METHOD FINAL metSave : BOOL
VAR_INPUT
    itfDataTypeObj  :   ITF_DATATYPE;
END_VAR
VAR
    uiSafetyCount   :   UINT;
    wPos            :   WORD;
    xSysSemapohre   :   BOOL;
END_VAR
IF proSave OR itfDataTypeObj.proSaveOnChange THEN  
    IF NOT itfDataTypeObj.proIsSaving THEN 
        itfDataTypeObj.proIsSaving := TRUE;
        xSysSemapohre := TRUE;   
    END_IF;
    IF xSysSemapohre THEN
        uiSafetyCount := 0;           
        REPEAT
            pResult := 0; 
            (* File Lesen *)
            IF NOT scState.xIsOpen THEN
                scState.xIsOpen := metOpenFile();
            END_IF;    
            IF scState.xIsOpen THEN
                metSave := metSaveFile(itfDataTypeObj);  
            END_IF;
            uiSafetyCount := uiSafetyCount + 1;
            IF NOT metSave THEN
                wPos := 16#EEEE;    
			END_IF
        UNTIL
            metSave = TRUE OR uiSafetyCount = 16#FFFF
        END_REPEAT
        IF NOT metSave THEN
            THIS^.proError      := TRUE;
            THIS^.proErrorNr    := itfDataTypeObj.proParaNr;
        END_IF  
        xSysSemapohre := FALSE;
        itfDataTypeObj.proIsSaving      := FALSE;
        itfDataTypeObj.proSaveOnChange  := FALSE;		
    END_IF;
END_IF;
END_METHOD

PROPERTY proError : BOOL
GET
proError := xError;
END_GET
SET
xError := proError;
END_SET
END_PROPERTY

{attribute 'monitoring_encoding' := 'UTF-8'}
PROPERTY proFilePath : STRING[255];
GET
// FILE Path auf SPS
proFilePath     :=      	CONCAT(
							CONCAT(
							CONCAT(                                
									'./',
									'ConfigFiles/Actual/'),
									stCodeDir),
									'_Config.txt');                                  
								
IF proLoad OR proSave THEN
	proFilePath     :=      CONCAT(
							CONCAT(
							CONCAT(    
							CONCAT(                            
									'./',
									'ConfigFiles/'),
									GVL_Config.stBackUp),
									stCodeDir),
									'_Config.txt');  
END_IF;
END_GET
END_PROPERTY

METHOD metCleanUpInit
VAR_INPUT
END_VAR
pResult     		:= fcFileClose(hFile,stCodeDir,'FbConfigFile CleanupIni Z1');
hFile       		:= 0;
pResultCheck		:= fcFileClose(hFileCheck,stCodeDir,'FbConfigFile CleanupIni Z3');
hFileCheck  		:= 0;
fcFileDelete(proFilePathCheckFile);
scState.xInit       := FALSE;
scState.xInitDone	:= TRUE;
iCaseInit   		:= iCaseInit + 1;
END_METHOD

METHOD FINAL metInit : BOOL
VAR_INPUT
    itfDataTypeObj  :   ITF_DATATYPE;
END_VAR
IF scstate.xGetChild THEN
	metChild(itfDataTypeObj);
END_IF;
IF scState.xInit THEN
    IF metCheckNr(itfDataTypeObj,TRUE,FALSE) THEN
        IF NOT metLoadFile(itfDataTypeObj) THEN
            metSaveFile(itfDataTypeObj);
        END_IF;  
        metCheckNr(itfDataTypeObj,FALSE,TRUE);
		metInit := TRUE;
    ELSE    
        proError    := TRUE;
        proErrorNr  := itfDataTypeObj.proParaNr;        
    END_IF;
	IF __QUERYINTERFACE(itfDataTypeObj,itfDataTypeObj) THEN
		IF itfDataTypeObj.proparaNr = usilastChild THEN
			metCleanUpInit();
		END_IF
	END_IF;         
END_IF;
END_METHOD

//FB_Init ist immer implizit verfügbar und wird primär für die Initialisierung verwendet.
//Der Rückgabewert wird nicht ausgewertet. Für gezielte Einflussnahme können Sie
//die Methoden explizit deklarieren und darin mit dem Standard-Initialisierungscode 
//zusätzlichen Code bereitstellen. Sie können den Rückgabewert auswerten.
METHOD FINAL FB_Init: BOOL
VAR_INPUT    
bInitRetains: BOOL; // TRUE: Die Retain-Variablen werden initialisiert (Reset warm / Reset kalt)    
bInCopyCode: BOOL;  // TRUE: Die Instanz wird danach in den Kopiercode kopiert (Online-Change)
END_VAR
hFile   := 0;
hFileCheck  := 0;
END_METHOD

{attribute 'monitoring':='call'}
PROPERTY proSave : BOOL
GET
proSave := GVL_Config.xSave;
END_GET
END_PROPERTY

{attribute 'monitoring':='call'}
PROPERTY proInitDone : BOOL
GET
proInitDone := scState.xInitDone;
END_GET
END_PROPERTY

PROPERTY ProSetInstancePathOnDynCreate : STRING(255)
SET
stCodeDir := ProSetInstancePathOnDynCreate;
metCodeDirCreate();
END_SET
END_PROPERTY

METHOD metCleanUp
VAR_INPUT	
END_VAR
pResult     		:= fcFileClose(hFile,stCodeDir,'FbConfigFile Cleanup Z1');
hFile       		:= 0;
scState.xIsOpen 	:= FALSE;
END_METHOD

METHOD metCheckLastChild
VAR_INPUT  
    itfDataTypeObj  :   ITF_DATATYPE;
END_VAR
IF __QUERYINTERFACE(itfDataTypeObj,itfDataTypeObj) THEN
	IF itfDataTypeObj.proparaNr = usilastChild THEN
		metCleanUp();
	END_IF
END_IF;
END_METHOD

END_FUNCTION_BLOCK

// 30 Program Organization Units/40 Byte String/fbSTRING40
FUNCTION_BLOCK fbSTRING40 EXTENDS fbDataType IMPLEMENTS ITF_STRING40
VAR_INPUT CONSTANT
	{attribute 'monitoring_encoding' := 'UTF-8'}
    _WertInit      :   STRING[40];  
END_VAR
VAR
	{attribute 'monitoring_encoding' := 'UTF-8'}
    stValue          :   STRING[40]; 
    {attribute 'hide'}
	{attribute 'monitoring_encoding' := 'UTF-8'}
    stValueOld       :   STRING[40]; 
END_VAR

(* Call Supper Objekt *)
IF itfConfigFb <> 0 THEN
    SUPER^();
END_IF;

{attribute 'hide'}
{attribute 'monitoring':='call'}
{attribute 'monitoring_encoding' := 'UTF-8'}
PROPERTY proStrPara : STRING(129)
// {attribute 'hide'}
GET
proStrPara :=   CONCAT(                    
                CONCAT( 
                CONCAT(
                CONCAT(                 
                CONCAT(                     
                CONCAT( fcfillStr(CONCAT('P',TO_STRING(SUPER^._usiParaNr)),6)       ,
                        ';'                                                         ),
                        fcfillStr(TO_STRING(stValue),GlobalKonstant.usiFeldLeng)    ),
                        ';'                                                         ),
                        fcfillStr('',GlobalKonstant.usiFeldLeng)                    ),
                        ';'                                                         ),
                        fcfillStr('',GlobalKonstant.usiFeldLeng)                    );
END_GET
SET
proValue  := fcGetValue(proStrPara);
END_SET
END_PROPERTY

METHOD metNewValueNoSave : BOOL
VAR_INPUT
    newValueNoSave   :   STRING[40];
END_VAR
proValue := newValueNoSave;
scState.xUpdateOldValueNoSave := TRUE;
metNewValueNoSave := TRUE;
END_METHOD

{attribute 'hide'}
METHOD metInit : BOOL
proValue  := _WertInit;
END_METHOD

{attribute 'monitoring_encoding' := 'UTF-8'}
PROPERTY proShowValue : STRING[40]
GET
proShowValue := stValue;
END_GET
END_PROPERTY

{attribute 'monitoring':='call'}
{attribute 'monitoring_encoding' := 'UTF-8'}
PROPERTY proValue : STRING[40]
SET
stValue := proValue;
(* Hack da Virtual Keyboard kein ° Zeichen hat *)
IF FIND(stValue,'§C') > 0 THEN
    stValue := REPLACE(stValue,'°',1,FIND(stValue,'§C'));
END_IF;
stValue[40] := 0;
END_SET
GET
stValue[40] := 0;
proValue := stValue;
END_GET
END_PROPERTY

METHOD metNewValue : BOOL
VAR_INPUT
    newValue   :   STRING[40];
END_VAR
proValue := newValue;
metNewValue := TRUE;
END_METHOD

{attribute 'hide'}
METHOD metCheckState : BOOL
(* Search Change & Save Old Values *)
IF stValue <> stValueOld OR scState.xUpdateOldValueNoSave THEN
    (* Prüfen ob die Werte bei änderung gespeichert werden sollen *)
    IF scState.xUpdateOldValueNoSave THEN
        scState.xUpdateOldValueNoSave := FALSE;
    ELSE
        proSaveOnChange 	:= TRUE;
	END_IF
	(*State Changed*) 
	scState.xStateChanged 	:= TRUE;   
    proValue 				:= stValue;
    stValueOld 				:= proValue;
ELSE
	(*State Changed*) 
	scState.xStateChanged 	:= FALSE;    
END_IF;
END_METHOD

END_FUNCTION_BLOCK

// 40 Visualizations/32 Bit/DWORD/visDWORD_QUERRY
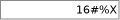
VISUALIZATION visDWORD_QUERRY  // 120x20
VAR_INPUT
    visfbDWORDIn :   ITF_DWORD;	
END_VAR
    Frame (0,0 120x20), invisible if: NOT __QUERYINTERFACE(visfbDWORDIn,visfbDWORDIn)
        shows visDWORD_ITF(visfbDWORD := visfbDWORDIn)
END_VISUALIZATION

// 40 Visualizations/1 Bit/visBOOL
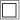
VISUALIZATION visBOOL  // 20x20
VAR_INPUT
    visfbBOOLIn  : ITF_DATATYPE;
END_VAR
VAR    
    visfbBOOL    : ITF_BOOL;    	
END_VAR
    Frame (0,0 20x20), invisible if: NOT __QUERYINTERFACE(visfbBOOLIn,visfbBOOL)
        shows visBOOL_QUERRY(visfbBOOLIn := visfbBOOL)
END_VISUALIZATION

// 40 Visualizations/32 Bit/UDINT/visUDINT
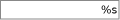
VISUALIZATION visUDINT  // 120x20
VAR_INPUT
    visfbUDINTIn :   ITF_DATATYPE;	
END_VAR
VAR
    visfbUDINT   :   ITF_UDINT;	
END_VAR
VAR_INPUT 
    stPhysikalischeEinheit  : STRING[5];
END_VAR
    Frame (0,0 120x20), invisible if: NOT __QUERYINTERFACE(visfbUDINTIn,visfbUDINT)
        shows visUDINT_QUERRY(visfbUDINTIn := visfbUDINT, stPhysikalischeEinheit := stPhysikalischeEinheit)
END_VISUALIZATION

// 40 Visualizations/32 Bit/TIME/visTIME
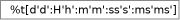
VISUALIZATION visTIME  // 180x20
VAR_INPUT   
    visfbTIMEIn :   ITF_DATATYPE;	
END_VAR
VAR  
    visfbTIME   :   ITF_TIME;	
END_VAR
    Frame (0,0 180x20), invisible if: NOT __QUERYINTERFACE(visfbTIMEIn,visfbTIME)
        shows visTIME_QUERRY(visfbTIMEIn := visfbTIME)
END_VISUALIZATION

// 40 Visualizations/32 Bit/REAL/visREAL_QUERRY
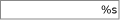
VISUALIZATION visREAL_QUERRY  // 120x20
VAR_INPUT    
    visfbREALIn :   ITF_REAL;	
END_VAR
VAR_INPUT 
    stPhysikalischeEinheit  : STRING[5];
END_VAR
    Frame (0,0 120x20), invisible if: NOT __QUERYINTERFACE(visfbREALIn,visfbREALIn)
        shows visREAL_ITF(visfbREAL := visfbREALIn, stPhysikalischeEinheit := stPhysikalischeEinheit)
END_VISUALIZATION

// 40 Visualizations/1 Bit/visBOOL_ITF
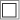
VISUALIZATION visBOOL_ITF  // 20x20
VAR_INPUT
    visfbBOOL    : ITF_BOOL;    	
END_VAR
    Checkbox (0,0 20x20), variable: visfbBOOL.proValue
END_VISUALIZATION

// 40 Visualizations/ENUMERATION/32 Bit/visENUMERATION_DINT_QUERRY
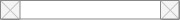
VISUALIZATION visENUMERATION_DINT_QUERRY  // 180x20
VAR_INPUT
    visfbDINT   :   ITF_DINT;	
END_VAR
    Frame (0,0 180x20), invisible if: NOT __QUERYINTERFACE(visfbDINT,visfbDINT)
        shows visENUMERATION_DINT(visfbDINT := visfbDINT)
END_VISUALIZATION

// 40 Visualizations/16 Bit/WORD/WORD HEX/visWORD_HEX
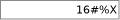
VISUALIZATION visWORD_HEX  // 120x20
VAR_INPUT
    visfbWORDIn :   ITF_DATATYPE;	
END_VAR
VAR
    visfbWORD   :   ITF_WORD;	
END_VAR
    Frame (0,0 120x20), invisible if: NOT __QUERYINTERFACE(visfbWORDIn,visfbWORD)
        shows visWORD_QUERRY_HEX(visfbWORDIn := visfbWORD)
END_VISUALIZATION

// 40 Visualizations/64 Bit/LTIME/visLTIME_ITF
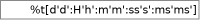
VISUALIZATION visLTIME_ITF  // 200x20
VAR_INPUT
    visfbLTIME   :   ITF_LTIME;	
END_VAR
    Textfield (0,0 200x20), "%t[d'd':H'h':m'm':ss's':ms'ms']", text variable: visfbLTIME.proValue
        OnMouseClick: write the text variable via InputWithLimits, min TO_ULINT(visfbLTIME.proMin), max TO_ULINT(visfbLTIME.proMax), title 'T#'
END_VISUALIZATION

// 40 Visualizations/32 Bit/REAL/visREAL
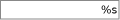
VISUALIZATION visREAL  // 120x20
VAR_INPUT
    visfbREALIn :   ITF_DATATYPE;	
END_VAR
VAR
    visfbREAL   :   ITF_REAL;	
END_VAR
VAR_INPUT 
    stPhysikalischeEinheit  : STRING[5];
END_VAR
    Frame (0,0 120x20), invisible if: NOT __QUERYINTERFACE(visfbREALIn,visfbREAL)
        shows visREAL_QUERRY(visfbREALIn := visfbREAL, stPhysikalischeEinheit := stPhysikalischeEinheit)
END_VISUALIZATION

// 40 Visualizations/32 Bit/DATE AND TIME/visDATE_AND_TIME_ITF
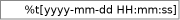
VISUALIZATION visDATE_AND_TIME_ITF  // 180x20
VAR_INPUT
    visfbDATE_AND_TIMEIn   :   ITF_DATE_AND_TIME;	
END_VAR
    Textfield (0,0 180x20), "%t[yyyy-mm-dd HH:mm:ss]", text variable: visfbDATE_AND_TIMEIn.proValue
        OnMouseClick: write the text variable via InputWithLimits, min TO_UDINT(visfbDATE_AND_TIMEIn.proMin), max TO_UDINT(visfbDATE_AND_TIMEIn.proMax), title 'T#'
END_VISUALIZATION

// 40 Visualizations/16 Bit/INT/visINT
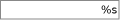
VISUALIZATION visINT  // 120x20
VAR_INPUT
    visfbINTIn :   ITF_DATATYPE;	
END_VAR
VAR
    visfbINT   :   ITF_INT;	
END_VAR
VAR_INPUT 
    stPhysikalischeEinheit  : STRING[5];
END_VAR
    Frame (0,0 120x20), invisible if: NOT __QUERYINTERFACE(visfbINTIn,visfbINT)
        shows visINT_QUERRY(visfbINTIn := visfbINT, stPhysikalischeEinheit := stPhysikalischeEinheit)
END_VISUALIZATION

// 40 Visualizations/32 Bit/UDINT/visUDINT_QUERRY
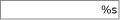
VISUALIZATION visUDINT_QUERRY  // 120x20
VAR_INPUT
    visfbUDINTIn :   ITF_UDINT;	
END_VAR
VAR_INPUT 
    stPhysikalischeEinheit  : STRING[5];
END_VAR
    Frame (0,0 120x20), invisible if: NOT __QUERYINTERFACE(visfbUDINTIn,visfbUDINTIn)
        shows visUDINT_ITF(visfbUDINT := visfbUDINTIn, stPhysikalischeEinheit := stPhysikalischeEinheit)
END_VISUALIZATION

// 40 Visualizations/8 Bit/SINT/visSINT_QUERRY
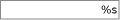
VISUALIZATION visSINT_QUERRY  // 120x20
VAR_INPUT
    visfbSINTIn :   ITF_SINT;	
END_VAR
VAR_INPUT 
    stPhysikalischeEinheit  : STRING[5];
END_VAR
    Frame (0,0 120x20), invisible if: NOT __QUERYINTERFACE(visfbSINTIn,visfbSINTIn)
        shows visSINT_ITF(visfbSINT := visfbSINTIn, stPhysikalischeEinheit := stPhysikalischeEinheit)
END_VISUALIZATION

// 40 Visualizations/16 Bit/WORD/WORD DEZ/visWORD_ITF_DEZ
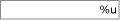
VISUALIZATION visWORD_ITF_DEZ  // 120x20
VAR_INPUT
    visfbWORD   :   ITF_WORD;	
END_VAR
    Textfield (0,0 120x20), "%u", text variable: visfbWORD.proValue
        OnMouseClick: write the text variable via InputWithLimits, min visfbWORD.proMin, max visfbWORD.proMax
END_VISUALIZATION

// 40 Visualizations/32 Bit/TOD/visTOD_ITF
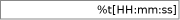
VISUALIZATION visTOD_ITF  // 180x20
VAR_INPUT
    visfbTODIn   :   ITF_TOD;	
END_VAR
    Textfield (0,0 180x20), "%t[HH:mm:ss]", text variable: visfbTODIn.proValue
        OnMouseClick: write the text variable via InputWithLimits, min TO_UDINT(visfbTODIn.proMin), max TO_UDINT(visfbTODIn.proMax), title 'Tod#'
END_VISUALIZATION

// 40 Visualizations/16 Bit/INT/visINT_ITF
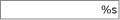
VISUALIZATION visINT_ITF  // 120x20
VAR_INPUT
    visfbINT   :   ITF_INT;	
END_VAR
VAR_INPUT 
    stPhysikalischeEinheit  : STRING[5];
END_VAR
    Textfield (0,0 120x20), "%s", text variable: CONCAT(TO_STRING(visfbINT.proValue),stPhysikalischeEinheit)
        OnMouseClick: write visfbINT.proValue via InputWithLimits, min visfbINT.proMin, max visfbINT.proMax
END_VISUALIZATION

// 40 Visualizations/8 Bit/USINT/visUSINT_QUERRY
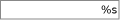
VISUALIZATION visUSINT_QUERRY  // 120x20
VAR_INPUT
    visfbUSINTIn :   ITF_USINT;	
END_VAR
VAR_INPUT 
    stPhysikalischeEinheit  : STRING[5];
END_VAR
    Frame (0,0 120x20), invisible if: NOT __QUERYINTERFACE(visfbUSINTIn,visfbUSINTIn)
        shows visUSINT_ITF(visfbUSINT := visfbUSINTIn, stPhysikalischeEinheit := stPhysikalischeEinheit)
END_VISUALIZATION

// 40 Visualizations/8 Bit/USINT/visUSINT_ITF
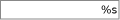
VISUALIZATION visUSINT_ITF  // 120x20
VAR_INPUT
    visfbUSINT   :   ITF_USINT;	
END_VAR
VAR_INPUT 
    stPhysikalischeEinheit  : STRING[5];
END_VAR
    Textfield (0,0 120x20), "%s", text variable: CONCAT(TO_STRING(visfbUSINT.proValue),stPhysikalischeEinheit)
        OnMouseClick: write visfbUSINT.proValue via InputWithLimits, min visfbUSINT.proMin, max visfbUSINT.proMax
END_VISUALIZATION

// 40 Visualizations/40 Byte String/visSTRING40_QUERRY
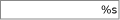
VISUALIZATION visSTRING40_QUERRY  // 120x20
VAR_INPUT
    visfbSTRING40In :   ITF_STRING40;	
END_VAR
    Frame (0,0 120x20), invisible if: NOT __QUERYINTERFACE(visfbSTRING40In,visfbSTRING40In)
        shows visSTRING40_ITF(visfbSTRING40In := visfbSTRING40In)
END_VISUALIZATION

// 40 Visualizations/16 Bit/WORD/WORD DEZ/visWORD_QUERRY_DEZ
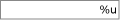
VISUALIZATION visWORD_QUERRY_DEZ  // 120x20
VAR_INPUT
    visfbWORDIn :   ITF_WORD;	
END_VAR
    Frame (0,0 120x20), invisible if: NOT __QUERYINTERFACE(visfbWORDIn,visfbWORDIn)
        shows visWORD_ITF_DEZ(visfbWORD := visfbWORDIn)
END_VISUALIZATION

// 40 Visualizations/40 Byte String/visSTRING40
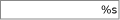
VISUALIZATION visSTRING40  // 120x20
VAR_INPUT
    visfbSTRING40In :   ITF_DATATYPE;	
END_VAR
VAR
    visfbSTRING40   :   ITF_STRING40;	
END_VAR
    Frame (0,0 120x20), invisible if: NOT __QUERYINTERFACE(visfbSTRING40In,visfbSTRING40)
        shows visSTRING40_QUERRY(visfbSTRING40In := visfbSTRING40)
END_VISUALIZATION

// 40 Visualizations/64 Bit/LTIME/visLTIME
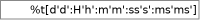
VISUALIZATION visLTIME  // 200x20
VAR_INPUT   
    visfbLTIMEIn :   ITF_DATATYPE;	
END_VAR
VAR  
    visfbLTIME   :   ITF_LTIME;	
END_VAR
    Frame (0,0 200x20), invisible if: NOT __QUERYINTERFACE(visfbLTIMEIn,visfbLTIME)
        shows visLTIME_QUERRY(visfbLTIMEIn := visfbLTIME)
END_VISUALIZATION

// 40 Visualizations/16 Bit/WORD/WORD DEZ/visWORD_DEZ
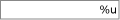
VISUALIZATION visWORD_DEZ  // 120x20
VAR_INPUT
    visfbWORDIn :   ITF_DATATYPE;	
END_VAR
VAR
    visfbWORD   :   ITF_WORD;	
END_VAR
    Frame (0,0 120x20), invisible if: NOT __QUERYINTERFACE(visfbWORDIn,visfbWORD)
        shows visWORD_QUERRY_DEZ(visfbWORDIn := visfbWORD)
END_VISUALIZATION

// 40 Visualizations/Show Data/visSHOWDATA_QUERRY
